(* Single tank with LimitSwitchLow (piLsLow) and LimitSwitchHigh (piLsHigh)
| using this function when it have INDEPENDENT Measure weight
*)
FUNCTION_BLOCK FB_SingleTankV1 EXTENDS FB_SingleTank
VAR
	bAllowInMaterial : BOOL;
	bAllowOutMaterial : BOOL;
	lrLimitMinWeight : LREAL;
	lrLimitMaxWeight : LREAL;
	lrWeightWithdraw : LREAL; 		// weight withdraw Request
	lrWeightBeforeWD : LREAL;
	lrWeightWithdrawN : LREAL;
	lrWeight : LREAL;
	eState : E_TankState;
	iFill : I_TankFill;				// the components that action for fill materials.
	
	tonRemainOffLsLow	: TON;
	tRemainOffLsLow	: TIME := T#1S;
	tonRemainLsHigh	: TON;
	tRemainLsHigh	: TIME := T#1S;	
	rTrigExecute : R_TRIG;
	bExecute : BOOL;//Execute with draw
	bFillError : BOOL;
	bError : BOOL;
END_VAR

SUPER^();
rTrigExecute(CLK := bExecute);
tonRemainOffLsLow(
	IN := NOT piLslow.In,
	PT := tRemainOffLsLow,
);
bAllowOutMaterial := (lrWeight > lrLimitMinWeight) AND NOT tonRemainOffLsLow.Q;

tonRemainLsHigh(
	IN := piLsHigh.In,
	PT := tRemainLsHigh,
);
bAllowInMaterial := (lrWeight < lrLimitMaxWeight) AND NOT tonRemainLsHigh.Q;
lrWeightWithdrawN := lrWeight-lrWeightBeforeWD;

CASE eState OF
	TANK_STOP:
		MS_Stop();
		
	TANK_WITHDRAWING:
		MS_Withdraw();
		
	TANK_FILLING:
		MS_Filling();
END_CASE

PROPERTY AllowIn : Reference to bool
GET
AllowIn ref= bAllowInMaterial;
END_GET
END_PROPERTY

(*
| Check the minimum condition  (lrWeight > lrLimitMinWeight
								AND piLslow.In;)
*)
PROPERTY AllowOut : REFERENCE TO BOOL
GET
AllowOut ref= bAllowOutMaterial;
END_GET
END_PROPERTY

METHOD AssignIfill : BOOL
VAR_INPUT
	iFill : I_TankFill;
END_VAR
THIS^.iFill := iFill;
END_METHOD

PROPERTY Error : reference to Bool
GET
Error ref= bError;
END_GET
END_PROPERTY

PROPERTY LimitMaxWeight : LREAL
GET
LimitMaxWeight := lrLimitMaxWeight;
END_GET
SET
lrLimitMaxWeight := LimitMaxWeight;
END_SET
END_PROPERTY

PROPERTY LimitMinWeight : LREAL
GET
LimitMinWeight := lrLimitMinWeight;
END_GET
SET
lrLimitMinWeight := LimitMinWeight;
END_SET
END_PROPERTY

METHOD MR_Filling : BOOL
VAR_INPUT
END_VAR
IF eState=TANK_STOP 
	AND bAllowInMaterial
THEN
	eState := TANK_FILLING;
END_IF
END_METHOD

METHOD MR_Reset : BOOL
VAR_INPUT
END_VAR
bError := FALSE;
MR_Reset := TRUE;
END_METHOD

METHOD MR_Stop : BOOL
VAR_INPUT
END_VAR
eState := TANK_STOP;
END_METHOD

(*	if withdrawing => still withdraw
	else
		if not stop => MR_Stop before withdraw
*)
METHOD MR_WithDraw : BOOL
VAR_INPUT
	lrWeightWd : LREAL;
	bExecute : BOOL;
END_VAR
THIS^.bExecute := bExecute;
IF rTrigExecute.Q
	AND eState=TANK_STOP 
	AND lrWeight > (lrWeightWd + lrLimitMinWeight) // Check enough weight
	AND bAllowOutMaterial
THEN
	eState := TANK_WITHDRAWING;
	lrWeightWithdraw := lrWeightWd;
	lrWeightBeforeWD := lrWeight;
END_IF
END_METHOD

METHOD PROTECTED MS_Filling
VAR_INPUT
END_VAR
IF bAllowInMaterial THEN
	iFill.Open();
ELSE
	iFill.Close();
	bError := TRUE;
	eState := TANK_STOP;
END_IF
END_METHOD

METHOD PROTECTED MS_Stop
VAR_INPUT
END_VAR
poCylinderCoil.Out := FALSE;
iFill.Close();
END_METHOD

METHOD PROTECTED MS_Withdraw
VAR_INPUT
END_VAR
poCylinderCoil.Out := TRUE;
IF lrWeightWithdrawN > lrWeightWithdraw THEN
	eState := TANK_STOP;
END_IF
IF NOT bAllowOutMaterial THEN
	bError := TRUE;
END_IF
END_METHOD

PROPERTY TimeRemainLsHigh : Time
GET
TimeRemainLsHigh := tRemainLsHigh;
END_GET
SET
tRemainLsHigh := TimeRemainLsHigh;
END_SET
END_PROPERTY

PROPERTY TimeRemainOffLsLow : Time
GET
TimeRemainOffLsLow := tRemainOffLsLow;
END_GET
SET
tRemainOffLsLow := TimeRemainOffLsLow;
END_SET
END_PROPERTY

PROPERTY Weight : lreal
GET
Weight := lrWeight;
END_GET
SET
Weight := lrWeight;
END_SET
END_PROPERTY

PROPERTY WeightWithdraw : lreal
GET
WeightWithdraw := lrWeightWithdraw;
END_GET
SET
lrWeightWithdraw := WeightWithdraw;
END_SET
END_PROPERTY

END_FUNCTION_BLOCK

(* stored: Version 1.1.0.1, ProductVersion 3.1.4024.12
   POU FB_SingleTankV1: Id {3c3c8172-9c8e-4f0e-8bd8-ee41f1a2ec87}, SpecialFunc None
   Folder MR: Id {5cf67c81-8cb5-4f7d-a783-6c3d30fd5008}
   Folder MS: Id {2d673f0c-5114-41d5-a648-da7c237cd1a2}
   Property AllowIn: Id {a5d1e9f2-1d23-4794-9392-8644ad8ab554}
   Get Get: Id {4611aad3-ae04-417a-8e61-b72d52a0c4c9}
   Property AllowOut: Id {5d4e6ea0-55ba-4704-a525-66ba75ae4a85}
   Get Get: Id {fa245f39-09b8-4716-b89c-489ebbbd1034}
   Method AssignIfill: Id {6bd1ecf2-a801-4d2d-a49e-ce6e70f9edd8}
   Property Error: Id {7ebab51c-a90a-4640-837f-1a05932ddb35}
   Get Get: Id {04299d28-0ce0-4d65-86b4-b62485ed6af6}
   Property LimitMaxWeight: Id {09fb551a-44f6-4d4c-a29c-9adbf53bc1cd}
   Get Get: Id {02401e58-0bb9-42a3-8fe1-495c415f6569}
   Set Set: Id {2848334a-9b22-45d2-ac30-3fd5e06e6022}
   Property LimitMinWeight: Id {92119500-b222-4856-9d65-fe07625525b9}
   Get Get: Id {67a0b6a7-533a-440e-a39d-a2e2b1939326}
   Set Set: Id {d4aabfd8-d758-407f-a9a5-9feeba1db405}
   Method MR_Filling: Id {675faff3-e06e-4478-bd66-fbd908bf06d7}
   Method MR_Reset: Id {b15a0cc9-b577-4d24-ac34-0685a159acfb}
   Method MR_Stop: Id {82b4db85-f8ed-4c20-8ca1-01f5e4e6426c}
   Method MR_WithDraw: Id {dedc9575-8cb4-4654-8401-576c6fa3352b}
   Method MS_Filling: Id {30f1ee8e-2a2f-403a-a94d-62ab4c64a6dc}
   Method MS_Stop: Id {b8da31e7-b431-43cd-8de9-5758288609be}
   Method MS_Withdraw: Id {338a2e54-065d-4b01-b9af-c195bfc8ff21}
   Property TimeRemainLsHigh: Id {eb2e0d34-edab-404c-a659-63569a9bd607}
   Get Get: Id {3cf94d45-a8a4-4ec1-a749-debac5b7f43a}
   Set Set: Id {abdff600-b92b-41a5-a64c-0ecd0d1bbda3}
   Property TimeRemainOffLsLow: Id {75350e51-91e4-4d30-b49a-1e01a3efea97}
   Get Get: Id {6f6ae728-e329-4428-8e6d-c8884c7fc6c6}
   Set Set: Id {0303e9e2-62c1-483d-af66-6d00db2542aa}
   Property Weight: Id {48882b1a-1508-4301-adb8-c089b6bbba6d}
   Get Get: Id {362c66b8-ca90-4246-a487-4309fe64b699}
   Set Set: Id {0ff9306f-3504-4a30-a76d-50375bef0eef}
   Property WeightWithdraw: Id {6d9ed7fc-1a86-4025-a41e-3fd4479388ad}
   Get Get: Id {1111ca0d-4b93-425c-9139-7bcae5615117}
   Set Set: Id {b23ab4a6-f158-435d-89cf-39a8467e5856} *)
